//     Box 71 (AT5100-0100)/DRV Statusword/Statusword <-> Data Pointer/Status
//     Box 71 (AT5100-0100)/DRV Target torque/Target torque <-> Data Pointer/Torque
//     Box 71 (AT5100-0100)/DRV Torque actual value/Torque actual value <-> Data Pointer/ActTorque
//     Box 71 (AT5100-0100)/XFB Inputs/Data <-> Data Pointer/HallSensorValues
//   (this object) <-> TcCOM Objects/XTS ProcessingUnit 1/XL Part 2/XL Module 50
//     Box 62 (AT5100-0100)/DRV Commutation angle/Commutation angle <-> Data Pointer/CommutationAngle
//     Box 62 (AT5100-0100)/DRV Controlword/Controlword <-> Data Pointer/Control
//     Box 62 (AT5100-0100)/DRV Statusword/Statusword <-> Data Pointer/Status
//     Box 62 (AT5100-0100)/DRV Target torque/Target torque <-> Data Pointer/Torque
//     Box 62 (AT5100-0100)/DRV Torque actual value/Torque actual value <-> Data Pointer/ActTorque
//     Box 62 (AT5100-0100)/XFB Inputs/Data <-> Data Pointer/HallSensorValues
//   (this object) <-> TcCOM Objects/XTS ProcessingUnit 1/XL Part 2/XL Module 51
//     Box 63 (AT5100-0100)/DRV Commutation angle/Commutation angle <-> Data Pointer/CommutationAngle
//     Box 63 (AT5100-0100)/DRV Controlword/Controlword <-> Data Pointer/Control
//     Box 63 (AT5100-0100)/DRV Statusword/Statusword <-> Data Pointer/Status
//     Box 63 (AT5100-0100)/DRV Target torque/Target torque <-> Data Pointer/Torque
//     Box 63 (AT5100-0100)/DRV Torque actual value/Torque actual value <-> Data Pointer/ActTorque
//     Box 63 (AT5100-0100)/XFB Inputs/Data <-> Data Pointer/HallSensorValues
//   (this object) <-> TcCOM Objects/XTS ProcessingUnit 1/XL Part 2/XL Module 52
//     Box 64 (AT5100-0100)/DRV Commutation angle/Commutation angle <-> Data Pointer/CommutationAngle
//     Box 64 (AT5100-0100)/DRV Controlword/Controlword <-> Data Pointer/Control
//     Box 64 (AT5100-0100)/DRV Statusword/Statusword <-> Data Pointer/Status
//     Box 64 (AT5100-0100)/DRV Target torque/Target torque <-> Data Pointer/Torque
//     Box 64 (AT5100-0100)/DRV Torque actual value/Torque actual value <-> Data Pointer/ActTorque
//     Box 64 (AT5100-0100)/XFB Inputs/Data <-> Data Pointer/HallSensorValues
//   (this object) <-> TcCOM Objects/XTS ProcessingUnit 1/XL Part 2/XL Module 53
//     Box 65 (AT5100-0100)/DRV Commutation angle/Commutation angle <-> Data Pointer/CommutationAngle
//     Box 65 (AT5100-0100)/DRV Controlword/Controlword <-> Data Pointer/Control
//     Box 65 (AT5100-0100)/DRV Statusword/Statusword <-> Data Pointer/Status
//     Box 65 (AT5100-0100)/DRV Target torque/Target torque <-> Data Pointer/Torque
//     Box 65 (AT5100-0100)/DRV Torque actual value/Torque actual value <-> Data Pointer/ActTorque
//     Box 65 (AT5100-0100)/XFB Inputs/Data <-> Data Pointer/HallSensorValues
//   (this object) <-> TcCOM Objects/XTS ProcessingUnit 1/XL Part 2/XL Module 54
//     Box 66 (AT5100-0100)/DRV Commutation angle/Commutation angle <-> Data Pointer/CommutationAngle
//     Box 66 (AT5100-0100)/DRV Controlword/Controlword <-> Data Pointer/Control
//     Box 66 (AT5100-0100)/DRV Statusword/Statusword <-> Data Pointer/Status
//     Box 66 (AT5100-0100)/DRV Target torque/Target torque <-> Data Pointer/Torque
//     Box 66 (AT5100-0100)/DRV Torque actual value/Torque actual value <-> Data Pointer/ActTorque
//     Box 66 (AT5100-0100)/XFB Inputs/Data <-> Data Pointer/HallSensorValues
//   (this object) <-> TcCOM Objects/XTS ProcessingUnit 1/XL Part 2/XL Module 55
//     Box 67 (AT5100-0100)/DRV Commutation angle/Commutation angle <-> Data Pointer/CommutationAngle
//     Box 67 (AT5100-0100)/DRV Controlword/Controlword <-> Data Pointer/Control
//     Box 67 (AT5100-0100)/DRV Statusword/Statusword <-> Data Pointer/Status
//     Box 67 (AT5100-0100)/DRV Target torque/Target torque <-> Data Pointer/Torque
//     Box 67 (AT5100-0100)/DRV Torque actual value/Torque actual value <-> Data Pointer/ActTorque
//     Box 67 (AT5100-0100)/XFB Inputs/Data <-> Data Pointer/HallSensorValues
//   (this object) <-> TcCOM Objects/XTS ProcessingUnit 1/XL Part 2/XL Module 56
//     Box 68 (AT5100-0100)/DRV Commutation angle/Commutation angle <-> Data Pointer/CommutationAngle
//     Box 68 (AT5100-0100)/DRV Controlword/Controlword <-> Data Pointer/Control
//     Box 68 (AT5100-0100)/DRV Statusword/Statusword <-> Data Pointer/Status
//     Box 68 (AT5100-0100)/DRV Target torque/Target torque <-> Data Pointer/Torque
//     Box 68 (AT5100-0100)/DRV Torque actual value/Torque actual value <-> Data Pointer/ActTorque
//     Box 68 (AT5100-0100)/XFB Inputs/Data <-> Data Pointer/HallSensorValues
//   (this object) <-> TcCOM Objects/XTS ProcessingUnit 1/XL Part 2/XL Module 57
//     Box 69 (AT5100-0100)/DRV Commutation angle/Commutation angle <-> Data Pointer/CommutationAngle
//     Box 69 (AT5100-0100)/DRV Controlword/Controlword <-> Data Pointer/Control
//     Box 69 (AT5100-0100)/DRV Statusword/Statusword <-> Data Pointer/Status
//     Box 69 (AT5100-0100)/DRV Target torque/Target torque <-> Data Pointer/Torque
//     Box 69 (AT5100-0100)/DRV Torque actual value/Torque actual value <-> Data Pointer/ActTorque
//     Box 69 (AT5100-0100)/XFB Inputs/Data <-> Data Pointer/HallSensorValues
//   (this object) <-> TcCOM Objects/XTS ProcessingUnit 1/XL Part 3/XL Module 1
//     Box 74 (AT5100-0100)/DRV Commutation angle/Commutation angle <-> Data Pointer/CommutationAngle
//     Box 74 (AT5100-0100)/DRV Controlword/Controlword <-> Data Pointer/Control
//     Box 74 (AT5100-0100)/DRV Statusword/Statusword <-> Data Pointer/Status
//     Box 74 (AT5100-0100)/DRV Target torque/Target torque <-> Data Pointer/Torque
//     Box 74 (AT5100-0100)/DRV Torque actual value/Torque actual value <-> Data Pointer/ActTorque
//     Box 74 (AT5100-0100)/XFB Inputs/Data <-> Data Pointer/HallSensorValues
//   (this object) <-> TcCOM Objects/XTS ProcessingUnit 1/XL Part 3/XL Module 2
//     Box 75 (AT5100-0100)/DRV Commutation angle/Commutation angle <-> Data Pointer/CommutationAngle
//     Box 75 (AT5100-0100)/DRV Controlword/Controlword <-> Data Pointer/Control
//     Box 75 (AT5100-0100)/DRV Statusword/Statusword <-> Data Pointer/Status
//     Box 75 (AT5100-0100)/DRV Target torque/Target torque <-> Data Pointer/Torque
//     Box 75 (AT5100-0100)/DRV Torque actual value/Torque actual value <-> Data Pointer/ActTorque
//     Box 75 (AT5100-0100)/XFB Inputs/Data <-> Data Pointer/HallSensorValues
//   (this object) <-> TcCOM Objects/XTS ProcessingUnit 1/XL Part 3/XL Module 3
//     Box 76 (AT5100-0100)/DRV Commutation angle/Commutation angle <-> Data Pointer/CommutationAngle
//     Box 76 (AT5100-0100)/DRV Controlword/Controlword <-> Data Pointer/Control
//     Box 76 (AT5100-0100)/DRV Statusword/Statusword <-> Data Pointer/Status
//     Box 76 (AT5100-0100)/DRV Target torque/Target torque <-> Data Pointer/Torque
//     Box 76 (AT5100-0100)/DRV Torque actual value/Torque actual value <-> Data Pointer/ActTorque
//     Box 76 (AT5100-0100)/XFB Inputs/Data <-> Data Pointer/HallSensorValues
//   (this object) <-> TcCOM Objects/XTS ProcessingUnit 1/XL Part 3/XL Module 4
//     Box 77 (AT5100-0100)/DRV Commutation angle/Commutation angle <-> Data Pointer/CommutationAngle
//     Box 77 (AT5100-0100)/DRV Controlword/Controlword <-> Data Pointer/Control
//     Box 77 (AT5100-0100)/DRV Statusword/Statusword <-> Data Pointer/Status
//     Box 77 (AT5100-0100)/DRV Target torque/Target torque <-> Data Pointer/Torque
//     Box 77 (AT5100-0100)/DRV Torque actual value/Torque actual value <-> Data Pointer/ActTorque
//     Box 77 (AT5100-0100)/XFB Inputs/Data <-> Data Pointer/HallSensorValues
//   (this object) <-> TcCOM Objects/XTS ProcessingUnit 1/XL Part 3/XL Module 46
//     Box 72 (AT5100-0100)/DRV Commutation angle/Commutation angle <-> Data Pointer/CommutationAngle
//     Box 72 (AT5100-0100)/DRV Controlword/Controlword <-> Data Pointer/Control
//     Box 72 (AT5100-0100)/DRV Statusword/Statusword <-> Data Pointer/Status
//     Box 72 (AT5100-0100)/DRV Target torque/Target torque <-> Data Pointer/Torque
//     Box 72 (AT5100-0100)/DRV Torque actual value/Torque actual value <-> Data Pointer/ActTorque
//     Box 72 (AT5100-0100)/XFB Inputs/Data <-> Data Pointer/HallSensorValues
//   (this object) <-> TcCOM Objects/XTS ProcessingUnit 1/XL Part 3/XL Module 47
//     Box 73 (AT5100-0100)/DRV Commutation angle/Commutation angle <-> Data Pointer/CommutationAngle
//     Box 73 (AT5100-0100)/DRV Controlword/Controlword <-> Data Pointer/Control
//     Box 73 (AT5100-0100)/DRV Statusword/Statusword <-> Data Pointer/Status
//     Box 73 (AT5100-0100)/DRV Target torque/Target torque <-> Data Pointer/Torque
//     Box 73 (AT5100-0100)/DRV Torque actual value/Torque actual value <-> Data Pointer/ActTorque
//     Box 73 (AT5100-0100)/XFB Inputs/Data <-> Data Pointer/HallSensorValues
//   (this object) <-> TcCOM Objects/XTS ProcessingUnit 1/XL Part 3/XL Module 5
//     Box 78 (AT5100-0100)/DRV Commutation angle/Commutation angle <-> Data Pointer/CommutationAngle
//     Box 78 (AT5100-0100)/DRV Controlword/Controlword <-> Data Pointer/Control
//     Box 78 (AT5100-0100)/DRV Statusword/Statusword <-> Data Pointer/Status
//     Box 78 (AT5100-0100)/DRV Target torque/Target torque <-> Data Pointer/Torque
//     Box 78 (AT5100-0100)/DRV Torque actual value/Torque actual value <-> Data Pointer/ActTorque
//     Box 78 (AT5100-0100)/XFB Inputs/Data <-> Data Pointer/HallSensorValues
//   (this object) <-> TcCOM Objects/XTS ProcessingUnit 1/XL Part 3/XL Module 6
//     Box 79 (AT5100-0100)/DRV Commutation angle/Commutation angle <-> Data Pointer/CommutationAngle
//     Box 79 (AT5100-0100)/DRV Controlword/Controlword <-> Data Pointer/Control
//     Box 79 (AT5100-0100)/DRV Statusword/Statusword <-> Data Pointer/Status
//     Box 79 (AT5100-0100)/DRV Target torque/Target torque <-> Data Pointer/Torque
//     Box 79 (AT5100-0100)/DRV Torque actual value/Torque actual value <-> Data Pointer/ActTorque
//     Box 79 (AT5100-0100)/XFB Inputs/Data <-> Data Pointer/HallSensorValues
//   (this object) <-> TcCOM Objects/XTS ProcessingUnit 1/XL Part 3/XL Module 7
//     Box 80 (AT5100-0100)/DRV Commutation angle/Commutation angle <-> Data Pointer/CommutationAngle
//     Box 80 (AT5100-0100)/DRV Controlword/Controlword <-> Data Pointer/Control
//     Box 80 (AT5100-0100)/DRV Statusword/Statusword <-> Data Pointer/Status
//     Box 80 (AT5100-0100)/DRV Target torque/Target torque <-> Data Pointer/Torque
//     Box 80 (AT5100-0100)/DRV Torque actual value/Torque actual value <-> Data Pointer/ActTorque
//     Box 80 (AT5100-0100)/XFB Inputs/Data <-> Data Pointer/HallSensorValues
//   (this object) <-> TcCOM Objects/XTS ProcessingUnit 1/XL Part 3/XL Module 8
//     Box 81 (AT5100-0100)/DRV Commutation angle/Commutation angle <-> Data Pointer/CommutationAngle
//     Box 81 (AT5100-0100)/DRV Controlword/Controlword <-> Data Pointer/Control
//     Box 81 (AT5100-0100)/DRV Statusword/Statusword <-> Data Pointer/Status
//     Box 81 (AT5100-0100)/DRV Target torque/Target torque <-> Data Pointer/Torque
//     Box 81 (AT5100-0100)/DRV Torque actual value/Torque actual value <-> Data Pointer/ActTorque
//     Box 81 (AT5100-0100)/XFB Inputs/Data <-> Data Pointer/HallSensorValues

// ---- DUTs/ST_MoverInfo.TcDUT
TYPE ST_MoverInfo :
STRUCT
	MoverOtcid : otcid;
	PlanarMoverCommandMode : MC_Planar_Mover_Command_Mode;
	State : MC_Planar_State;
	Positition : LREAL;
	Track : Otcid;
	Error: BOOL;
	ErrorID : UDINT;
	TargetTrackPosition  : LREAL;
	TargetTrack : Otcid;
	RemainingDistance : LREAL;
	Gap : LREAL;
	LimitVelo : LREAL; 
	LimitAcc : LREAL;
	LimitDec : LREAL;
	LimitJerk : LREAL;
	
END_STRUCT
END_TYPE

// ---- DUTs/ST_MoverOnTrackInfo.TcDUT
TYPE ST_MoverOnTrackInfo :
STRUCT
	TargetPosition 		: LREAL;
	TargetTrack 		: Otcid;
	Remainingdistance 	: LREAL;
	Gap 				: LREAL;
	LimitV 				: LREAL;
	LimitA 				: LREAL;
	LimitD 				: LREAL;
	LimitJ 				: LREAL;
	GapMode				: MC.MC_GAP_MODE_ON_TRACK;
	DynamicMode			: MC.MC_DYNAMIC_MODE_ON_TRACK;
	Movementtype		: MC.MC_MOVEMENT_TYPE_ON_TRACK;
	
END_STRUCT
END_TYPE

// ---- XlMover/ITFs/I_Mover.TcIO

INTERFACE I_Mover

METHOD CycleUpdate : BOOL
VAR_INPUT
END_VAR
END_METHOD

PROPERTY distToEndOfTrack : Lreal
GET
END_GET
END_PROPERTY

METHOD Init : BOOL
VAR_INPUT
	XtsMover:  I_XtsXlMover1;
	XtsProcessingUnit :  I_XtsProcessingUnit1;
END_VAR
END_METHOD

METHOD JoinNearestTrack : BOOL


VAR

END_VAR
END_METHOD

METHOD LeaveSystemAt : BOOL
VAR_INPUT
	ConnectionOut: REFERENCE TO MC_PlanarTrackConnectionOut;	
END_VAR
END_METHOD

METHOD MoveOnTrack : BOOL
VAR_INPUT
	track: REFERENCE TO MC_PlanarTrack;	
	targetPos: LREAL;
	gap : LREAL; 

END_VAR
END_METHOD

PROPERTY MoverOTCID : OTCID
GET
END_GET
SET
END_SET
END_PROPERTY

PROPERTY MoverStopped : BOOL
GET
END_GET
SET
END_SET
END_PROPERTY

PROPERTY P_Dynamics : REFERENCE TO DynamicConstraint_PathXY;
GET
END_GET
END_PROPERTY

PROPERTY P_IsInitialized : bool
GET
END_GET
END_PROPERTY

PROPERTY P_PlanarFeedback : REFERENCE TO MC_PlanarFeedback
GET
END_GET
END_PROPERTY

PROPERTY P_PlanarMover :   REFERENCE TO  MC_PlanarMover
GET
END_GET
END_PROPERTY

PROPERTY P_SyncFeedback :  REFERENCE TO MC_PlanarFeedbackGearInPosOnTrackWithMasterMover
GET
END_GET
END_PROPERTY

PROPERTY P_TargetTrack : UDINT
GET
END_GET
SET
END_SET
END_PROPERTY

PROPERTY Rework : BOOL
GET
END_GET
SET
END_SET
END_PROPERTY

METHOD SyncToOtherMover : Bool
VAR_INPUT
	masterSyncPos : LREAL; // Position on the master track
	followerSyncPos : LREAL; // position on the follower track
	PlanarMoverToFollow: REFERENCE TO Tc3_Mc3PlanarMotion.MC_PlanarMover;
	masterTrack : REFERENCE TO Tc3_Mc3PlanarMotion.MC_PlanarTrack; 
	followerTrack : REFERENCE TO Tc3_Mc3PlanarMotion.MC_PlanarTrack; 
	velo :  REFERENCE TO LREAL; 
END_VAR
END_METHOD

METHOD  UpdateXtsTrack
VAR_INPUT
END_VAR
VAR

END_VAR
END_METHOD

PROPERTY XlProcessingUnit : I_XtsProcessingUnit1
GET
END_GET
END_PROPERTY

PROPERTY XtsComFeed : REFERENCE TO  XtsCommandFeedback
GET
END_GET
END_PROPERTY

PROPERTY XtsXlMover :  I_XtsXlMover1
GET
END_GET
END_PROPERTY

END_INTERFACE

// ---- POUs/FB_TrackObject.TcPOU
FUNCTION_BLOCK FB_TrackObject
// for a track/part this block keeps a list of the movers in order with their positions on a track

VAR_INPUT
	TrackID: OTCID;
	iMover	:REFERENCE TO ARRAY[1..nMoverCount] OF I_Mover;
END_VAR

VAR_OUTPUT
	bBusy: BOOL;
	bDone: BOOL;
	bError: BOOL;
	bInit: BOOL;
	ipResultMessage: I_TcMessage := fbResult;
	moverIDs : ARRAY[1..nMoverCount] OF UDINT;
	
END_VAR

VAR_STAT
	nNumMoversOnTrack: UDINT; //numberofMovers currently on this track
	nMoverList: ARRAY [1..nMoverCount] OF OTCID; //list of movers currently on the track 
	
	Moverdist: ARRAY[1..nMoverCount] OF LREAL;
	MoverPos: ARRAY[1..nMoverCount] OF LREAL;
	
	
END_VAR

VAR

	fbResult: FB_TcMessage;
	_ipComObject: ITComObject;
	PID_MOverList				: PTCID := 16#05030149;
	PID_NumMover				: PTCID := 16#050300C5;
END_VAR

IF NOT bInit THEN
	IF GetComObject(nObjectId:=TrackID) THEN
		bInit:=TRUE;
	END_IF
	RETURN;
END_IF

METHOD CyclicUpdate : BOOL
VAR_INPUT
END_VAR

VAR_INST
	J: UDINT;
	I: UINT;
END_VAR
IF bInit THEN 
	GetNumMovers(); 
	GetMoverList(); 
END_IF 
MEMSET(ADR(moverIDs),0,SIZEOF(moverIDs)); // have to clear the list 
MEMSET(ADR(Moverdist),0,SIZEOF(Moverdist)); // have to clear the list 
MEMSET(ADR(MoverPos),0,SIZEOF(MoverPos)); // have to clear the list 
FOR J := 1 TO nNumMoversOnTrack DO  
	FOR I := 1 TO nNumMovers DO  
		IF iMover[I].MoverOTCID = nMoverList[J] THEN 
			moverIDs[J] := I; 
		END_IF
	END_FOR

	
END_FOR

FOR J := 1 TO nNumMoversOnTrack DO  
	
	IF J < nNumMoversOnTrack - 1 THEN 
		 IF fbMover[moverIDs[j+1]].distToEndOfTrack - fbMover[moverIDs[j]].distToEndOfTrack > 0 THEN 
			Moverdist[j]:= fbMover[moverIDs[j+1]].distToEndOfTrack - fbMover[moverIDs[j]].distToEndOfTrack;
		ELSE
			Moverdist[j]:=-1;	
		END_IF
		MoverPos[j]:= fbMover[moverIDs[j+1]].distToEndOfTrack; // folowwing movers distance 
		//idist := fbMover[moverIDs[I]].distToEndOfTrack; //this movers distance 
	END_IF
	
END_FOR
END_METHOD

METHOD findMergePosition : BOOL
VAR_INPUT
	mergeSyncCommandPos : LREAL;
	spaceToMerge :LREAL; 
END_VAR
VAR_OUTPUT 
	nMoverToFollow: UDINT; 
	mergeWithoutFollow : BOOL; 
	mergeNotPossible : BOOL; 
END_VAR
VAR_INST 
	I: UDINT;
	moverInMerge: UDINT;
	moverIsWhereWeSync: BOOL;
	moversDist: LREAL;
	Iplus1Dist: LREAL;
	idist: LREAL;

	needToFollow: BOOL;

END_VAR
mergeNotPossible := TRUE; 
mergeWithoutFollow:=FALSE;
nMoverToFollow := 0; 
moverInMerge := 0;
needToFollow := TRUE;  
IF nNumMoversOnTrack = 0  THEN // if there's no movers on the track we can just merge 
	mergeWithoutFollow := TRUE;
	mergeNotPossible := FALSE; 
ELSE
  	// there's movers in the track we need to look where there are 
	// go through the movers positions and find a place to merge if available 
	FOR I := 1 TO nNumMoversOnTrack DO 
		// is this mover in the range where we would sync? 
		moverIsWhereWeSync := IsBetween(fbMover[moverIDs[I]].distToEndOfTrack, mergeSyncCommandPos, mergeSyncCommandPos + spaceToMerge); 
		needToFollow := IsBetween(fbMover[moverIDs[I]].distToEndOfTrack, mergeSyncCommandPos, mergeSyncCommandPos + spaceToMerge); //lagerwindow we can merge but must sync still
		IF moverIsWhereWeSync THEN //if the mover is where we would sync start looking for places to merge behind it
			moverInMerge := moverIDs[I]; // this mover is is the id of the mover thats in the way 
			// can we merge behind this one ?
			IF I < nNumMoversOnTrack THEN 
		//		Moverdist[i+10]:=moversDist := fbMover[moverIDs[I+1]].distToEndOfTrack - fbMover[moverIDs[I]].distToEndOfTrack;
	//			Moverdist[i]:=Iplus1Dist := fbMover[moverIDs[I+1]].distToEndOfTrack; // folowwing movers distance 
	//			idist := fbMover[moverIDs[I]].distToEndOfTrack; //this movers distance 
				// is the spacing between these two movers bigger than the space we need to merge?
				IF (Moverdist[i] )> spaceToMerge THEN 
					nMoverToFollow := moverIDs[I]; //yes follow this mover 
					mergeNotPossible := FALSE; // the merge is possible 
					EXIT; 
				END_IF
			ELSIF I = nNumMoversOnTrack THEN // this is the last mover 
				// look how much space is behind this mover that is bigger than the merge gap, merge behind this mover
				IF fbMover[moverIDs[I]].distToEndOfTrack < mergeSyncCommandPos+spaceToMerge THEN // the mover is far enough along to sync to it.
					nMoverToFollow := moverIDs[I]; //yes follow this mover 
					mergeNotPossible := FALSE; // the merge is possible 
				END_IF  
			END_IF	
		END_IF
	END_FOR 
	//if we went through the whole list and no mover is in the range where we would merge in, then just merge 
	IF fbMover[moverIDs[1]].distToEndOfTrack > 6000 THEN //there's noone where we want to merge, just merge in 
		mergeWithoutFollow:=TRUE;
		mergeNotPossible := FALSE;
	END_IF
END_IF
IF mergeNotPossible THEN 
	nMoverToFollow := 0; 
END_IF
END_METHOD

METHOD GetComObject : BOOL
VAR_INPUT
	nObjectId: OTCID;
END_VAR
IF FW_ObjMgr_GetObjectInstance(	oid		:= nObjectId, 
								iid		:= TC_GLOBAL_IID_LIST.IID_ITComObject, 
								pipUnk	:= ADR(_ipComObject)) = 0
THEN
	GetComObject := TRUE;
END_IF
END_METHOD

METHOD GetMoverList : BOOL
VAR
	nData 			: UDINT := SIZEOF(nMoverList);
	pData 			: PVOID := ADR(nMoverList);
	stEventEntry	: TcEventEntry;
	pstEventEntry	: REFERENCE TO TcEventEntry REF= stEventEntry;
END_VAR
VAR_INST
	hResult : HRESULT;
END_VAR
bError := FALSE;

IF _ipComObject <> 0 THEN 
	 hResult := 	_ipComObject.TcgetObjPara(		pid := PID_MOverList,
													nData := nData,
													pData := pData,
													pgp := 0); 	
	IF hResult = 0 THEN
		GetMoverList := TRUE;
	ELSE
		HRESULTAdsErr_TO_TcEventEntry(hResult,stEventEntry);
		IF NOT fbResult.EqualsToEventEntryEx( stOther := stEventEntry) THEN
			fbResult.CreateEx(stEventEntry, 0);
			fbResult.Send(0);
			fbResult.Release();
		END_IF
		bError := TRUE;
	END_IF							
END_IF
END_METHOD

METHOD GetNumMovers : BOOL
VAR
	stEventEntry: TcEventEntry;
	pstEventEntry: REFERENCE TO TcEventEntry := stEventEntry;
	nData 			: UDINT := SIZEOF(nNumMoversOnTrack);
	pData 			: PVOID := ADR(nNumMoversOnTrack);
END_VAR

VAR_INST
	hResult : HRESULT;
END_VAR
bError := FALSE;

IF _ipComObject <> 0 THEN 	
	

	 hResult := 	_ipComObject.TcGetObjPara(		pid := PID_NumMover,
													nData := nData,
													pData := pData,
													pgp := 0); 	
	IF hResult = 0 THEN
		GetNumMovers := TRUE;
	ELSE
		HRESULTAdsErr_TO_TcEventEntry(hResult,stEventEntry);
		IF NOT fbResult.EqualsToEventEntryEx( stOther := stEventEntry) THEN
			fbResult.CreateEx(stEventEntry, 0);
			fbResult.Send(0);
			fbResult.Release();
		END_IF
		bError := TRUE;
	END_IF							
END_IF
END_METHOD

END_FUNCTION_BLOCK

// ---- POUs/MAIN.TcPOU
PROGRAM MAIN
VAR
	RuntimeDuration	: STRING;
	TempRuntimeDur	: TIME;
	RuntimeTimer	: TON;
	CurrentSysTime	: ULINT;

	bAllDone		: BOOL;
	bStopSequence	: BOOL;
	HMI_StopCmd		: BOOL;
	
	nCase 		: INT;
	nMoveState		: ARRAY[1..nMoverCount] OF INT;
	

	
	nForCounter: UDINT;
	M,N,T,Tr : UINT;
//	slowDynamics: DynamicConstraint_PathXY;
	haltDynamics : DynamicConstraint_PathXY;
	stopAndWait : ARRAY[1..GVL_Mc.nMoverCount] OF TON; 
	waitForGapParkPos: LREAL := 3500;
	// Magnet
	MagnetValue AT%Q*: INT;
	MagnetFdbkValue AT%I* : INT;
	bMagnetOn : BOOL;
	MagnetOnManHMICmd 	: BOOL;
	tMagnetOnTime	: TIME := T#3S;

	Init : BOOL ; 	
	
	IsMoverCommandedInShortcut: BOOL;
	IsMoverInBlockingArea: BOOL;
	nActStopPos: UINT := 1;
	Fp_error : R_Trig;

	Switch : BOOL;
	WithoutSwitch : BOOL := TRUE;
	SwtichOnly: BOOL;
	
	MoverStop 	AT%I* :BOOL;
	MoverStopDone AT%Q*		: BOOL;
	Info 		AT%Q*: BOOL;
	Operating	AT%Q*: BOOL;
	Process		AT%Q*: BOOL;
	Fault		AT%Q*: BOOL;
	Emergency	AT%Q*: BOOL;
	
	Voltage1 AT%I*: UDINT;
	Voltage2 AT%I*: UDINT;
	
	
	TcRestart : TC_Restart;
	Restart : BOOL;
	busy : BOOL;
	rt_InitStart : R_TRIG;
	rt_InitStop : R_TRIG;
	bStartSequence: BOOL;
	
	FP_Counter : r_trig;
	Switchcounter : DINT;
	test : LREAL;
	Horntimer : tp; 
	R_trigHorn : R_trig;
	
	TestPowerMat : BOOL := TRUE;
	StopTime : TIME := T#1S;
	StopTimer :ARRAY[1..nMoverCount] OF ton;
	StartTimer :ARRAY[1..nMoverCount] OF BOOL;
	
	
	MoverPos :ARRAY[1..nMoverCount] OF PositionXYC;
	ArcLength :ARRAY[1..nMoverCount] OF LREAL;
	TrackPos :ARRAY[1..nMoverCount] OF ARRAY[1..nMoverCount] OF PositionXYC;
	
	//searchGap : F_SearchTheBigTrackForAHole; 
	aMoverTrack : ARRAY[1..nMoverCount] OF Global.OTCID;
	FirstMoverTrackPos : LREAL;
	MoverGap : LREAL;
	FTrigTrackCount : F_Trig;
	MoverNo  : UDINT;
	stMoverConfigSlow	: ST_MoverConfig;
	stMoverConfigNormal : ST_MoverConfig;
	stMoverConfigFast  : ST_MoverConfig;
	stMoverCfgAggressive : ST_MoverConfig;
	stMoverCfgHalt : ST_MoverConfig;
	
	stMergeConfig		 : ST_MergeConfig;
	SwitchConfig		 : ST_SwitchConfig;
	
	SwitchStatus 		  : ST_SwitchStatus;

	ModuleState1 AT%I*: E_EcState;
	ModuleState2 AT%I*: E_EcState;
	ModuleState3 AT%I*: ARRAY[0..2] OF E_EcState;
	
	MessageTrigger : ARRAY[1..20] OF R_trig;
	
	//========= Merge =========================================
	
	SwitchParkPos : LREAL := 3500;
	nextMoverForSwitch: UDINT :=1;
	moverInSwitchDoNotSendAnother: BOOL;
	trapError: BOOL;
	trapErrorID: UDINT;
	moverWithFault: UDINT;
	stepWithFault: INT;
	
	followSyncPos: LREAL;
	masterSyncPos: LREAL;
	masterPosAtSync: LREAL;
	followerPosAtSync: LREAL;
	moverInFront: UDINT;
	gapStart: LREAL := 8500; //5600
	gapLength: LREAL := 2200; //1800
	fbTrackobject : FB_TrackObject;
	getList: BOOL;
	directMerge: BOOL;
	mergeNotPossible: BOOL;
	
	endOfBigTrack : LREAL; 
	endOfSmallTrack : LREAL; 
	endOfMainTrack : LREAL; 
	followerToEndOfTrack: LREAL;
	leaderToEndofTrack: LREAL;
	distToMoverInFront: LREAL;
	moverSwitching: UDINT;
	switchingMoverPosition: LREAL;
	trapWhenMagnetturnedOn: R_TRIG;
	moverPositionWhenMagnetTurnedOn: LREAL;
	moverInSwitch: UDINT;
END_VAR


// =====================
// Initalize XTS Utility
GVL_MC.fbXtsEnvironment.Init(GVL_MC.cmdFeedback);
IF NOT GVL_MC.cmdFeedback.IsDone THEN
	RETURN;
END_IF
//*****************************************************
Emergency :=  MoverStop;

Operating := NOT  MoverStop;

//================== Check Voltage=====================================================
R_trigHorn(clk := Voltage1< 250000 );
//Horntimer(in:= ( R_trigHorn.Q ) , PT:= T#2S,Q=> info);
IF R_trigHorn.Q THEN
	ADSLOGSTR(msgCtrlMask:= ADSLOG_MSGTYPE_LOG , msgFmtStr:= 'Module Voltage Fault ' , strArg:= '');
END_IF 
//=================== Check State of Modules===========================================

MessageTrigger[1](clk:=ModuleState1 <> 8 AND nCASE> 0);
IF MessageTrigger[1].Q THEN
	ADSLOGSTR(msgCtrlMask:= ADSLOG_MSGTYPE_LOG , msgFmtStr:= 'Module Fault Line 1 %s' , strArg:= TO_STRING(ModuleState1));
END_IF

MessageTrigger[2](clk:=ModuleState2 <> 8 AND nCASE> 0);
IF MessageTrigger[2].Q THEN
	ADSLOGSTR(msgCtrlMask:= ADSLOG_MSGTYPE_LOG , msgFmtStr:= 'Module Fault Line 2 %s ' , strArg:= TO_STRING(ModuleState2));
END_IF

MessageTrigger[3](clk:=ModuleState3[0] <> 8 AND nCASE> 0);
IF MessageTrigger[3].Q THEN
	ADSLOGSTR(msgCtrlMask:= ADSLOG_MSGTYPE_LOG , msgFmtStr:= 'Module Fault Line 3 Default SyncUnit %s ' , strArg:= TO_STRING(ModuleState3[0]));
END_IF

MessageTrigger[4](clk:=ModuleState3[1] <> 8 AND nCASE> 0);
IF MessageTrigger[4].Q THEN
	ADSLOGSTR(msgCtrlMask:= ADSLOG_MSGTYPE_LOG , msgFmtStr:= 'Module Fault Line 3 XtsTask SyncUnit %s ' , strArg:= TO_STRING(ModuleState3[1]));
END_IF

MessageTrigger[5](clk:=ModuleState3[2] <> 8 AND nCASE> 0);
IF MessageTrigger[5].Q THEN
	ADSLOGSTR(msgCtrlMask:= ADSLOG_MSGTYPE_LOG , msgFmtStr:= 'Module Fault Line 3 PlcTask SyncUnit %s ' , strArg:= TO_STRING(ModuleState3[2]));
END_IF

//=====================================================================================

IF nCASE > 90 THEN
	Process := TRUE;
ELSE 
	Process := FALSE;	
END_IF

IF NOT MoverStop AND NOT MoverStopDone AND (nCase = 100) THEN
	ADSLOGSTR(msgCtrlMask:= ADSLOG_MSGTYPE_LOG , msgFmtStr:= 'E-Stop ' , strArg:= '');
	FOR nForCounter:=1 TO nNumMovers DO
		fbMover[nForCounter].P_Dynamics.SetValuesVADJ(stMoverConfigNormal.velo,stMoverConfigNormal.Accel,stMoverConfigNormal.Decel,stMoverConfigNormal.Jerk);
		nCase := 140;
	END_FOR		
ELSIF 	MoverStop THEN
	MoverStopDone := FALSE;
END_IF



TcRestart(
NETID:= '', 
RESTART:= Restart OR (GVL_Mc.HWStart AND NOT GVL_Mc.HWStop), 
TMOUT:=T#5S , 
BUSY=>busy , 
ERR=> , 
ERRID=> );

CurrentSysTime	:= Tc2_System.F_GetSystemTime();

IF TcRestart.BUSY THEN
	RuntimeTimer.IN 	:= FALSE;
ELSIF Process THEN
	RuntimeTimer.IN		:= TRUE;
	TempRuntimeDur		:= RuntimeTimer.ET;
	RuntimeDuration		:= TIME_TO_STRING(TempRuntimeDur);
END_IF
RuntimeTimer(PT := T#7D);

rt_InitStart(clk:= (bStartSequence OR GVL_Mc.HWStart) AND GVL_Mc.HWStop);
IF rt_InitStart.Q THEN
	nCase := 10;
	bStartSequence	:= FALSE;

	stMoverConfigSlow.Velo := 1000;
// 	stMoverConfigSlow.Accel := 4000;
// 	stMoverConfigSlow.Decel := 4000; 
// 	stMoverConfigSlow.Jerk := 16000;
	stMoverConfigFast.Velo := 4000;
// 	stMoverConfigFast.Accel := 4000;
// 	stMoverConfigFast.Decel := 4000; 
// 	stMoverConfigFast.Jerk := 16000;
	stMoverCfgHalt.Decel := 2000; 
	stMoverCfgHalt.Jerk := 10000;
	
//	slowDynamics.SetValuesVADJ(stMoverConfigSlow.Velo,stMoverConfigSlow.Accel,stMoverConfigSlow.Decel,stMoverConfigSlow.Jerk);
//	fastDynamics.SetValuesVADJ(stMoverConfigFast.Velo,stMoverConfigFast.Accel,stMoverConfigFast.Decel,stMoverConfigFast.Jerk);
	haltDynamics.SetValuesVADJ(stMoverCfgHalt.Velo,stMoverCfgHalt.Accel,stMoverCfgHalt.Decel,stMoverCfgHalt.Jerk);
END_IF
haltDynamics.SetValuesVADJ(stMoverCfgHalt.Velo,stMoverCfgHalt.Accel,stMoverCfgHalt.Decel,stMoverCfgHalt.Jerk);
GVL_Mc.StartLight := MoverStop AND nCase < 100;
GVL_Mc.StopLight  := (nCase = 100);

IsMoverInBlockingArea := FALSE;

FOR M := 1 TO GVL_Mc.nNumMovers DO///Movers
	StopTimer[M](in:=StartTimer[m],PT:=StopTime);

	
	IF NOT GVL_MC.fbMover[GVL_Mc.nNumMovers].P_IsInitialized THEN
		GVL_MC.ipXtsProcessingUnit :=  GVL_MC.fbXtsEnvironment.ProcessingUnit(1,0);
		GVL_MC.ipXlMover  :=  GVL_MC.fbXtsEnvironment.ProcessingUnit(1, 0).XlMover(m, 0);
		GVL_MC.fbMover[m].Init( GVL_MC.ipXlMover, GVL_MC.ipXtsProcessingUnit); 
		iMover[m] := fbMover[m] ;
	END_IF
	 MoverFeedback[m].Update();
	GVL_MC.fbMover[m].CycleUpdate();
	
	GVL_Mc.Mover[M].MoverPos  :=GVL_MC.fbMover[M].P_PlanarMover.MCTOPLC.SETONTRACK.SetPos;
	GVL_Mc.Mover[M].TrackID:= GVL_MC.fbMover[M].P_PlanarMover.MCTOPLC.SETONTRACK.TrackOID;
	GVL_Mc.Mover[M].MoverNumber := M;
		
	TR := Tr+1;
	IF Tr = 4 THEN
		Tr :=1;
	END_IF
	ArcLength[M] :=GVL_Mc.MC_Tracks[Tr].GetArcLengthClosestTo(MoverPos[M]);
	GVL_Mc.MC_Tracks[Tr].GetPositionAt(ArcLength[M],TrackPos[M][Tr]);
	
	IF ABS(MoverPos[m].x - TrackPos[M][Tr].x) < 1 AND  ABS(MoverPos[m].y - TrackPos[M][Tr].y) < 1 THEN
 		GVL_Mc.Mover[M].MoverTrackNr := Tr;
	END_IF	
	
	IsMoverInBlockingArea := IsMoverInBlockingArea OR (Mover[M].TrackID = GVL_Mc.MC_Tracks[E_TrackNum.main].MCTOPLC_STD.TrackOID AND IsBetween(Mover[M].MoverPos, SwitchConfig.MagnetStartPosition - 100, SwitchConfig.MagnetEndPosition + 100));

	Fp_error(clk := GVL_MC.fbMover[M].P_PlanarMover.Error AND GVL_MC.fbMover[M].XtsXlMover.GetIsActive(0) AND nCASE = 100);
	IF Fp_error.Q THEN
		nCase := 140;
		Fault := TRUE;
		bMagnetOn := FALSE;
		ADSLOGSTR(msgCtrlMask:= ADSLOG_MSGTYPE_LOG , msgFmtStr:= 'Mover %s Faulted ' , strArg:= INT_TO_STRING(M));
	ELSE
		Fault := FALSE;
	END_IF
	
	IF aMoverTrack[1] <> 0 AND_THEN GVL_MC.fbMover[M].P_PlanarMover.MCTOPLC.STD.MoverOID = aMoverTrack[1] THEN
		FirstMoverTrackPos := GVL_MC.fbMover[M].P_PlanarMover.MCTOPLC.SETONTRACK.SetPos;
	END_IF
	
END_FOR

FOR T := 1 TO nTrackCount DO 
	MC_Tracks[T].Update();
	MC_Trackfeedback[T].Update();
	
END_FOR
 MoverGap := (GVL_Mc.MC_Tracks[E_TrackNum.Big].GetLength()- FirstMoverTrackPos);
 
//================  merge ===============

fbTrackobject(TrackID:= MC_Tracks[E_TrackNum.big].MCTOPLC_STD.TrackOID,iMover:= iMover,trackLength:= GVL_Mc.MC_Tracks[E_TrackNum.Big].GetLength()); 
fbTrackobject.CyclicUpdate(); 


//======================================

CASE nCase OF
	10:
		
		Fault := FALSE;
		nCase := 20;

	20:
		FOR T := 1 TO nTrackCount DO 
			MC_Tracks[T].Enable(MC_Trackfeedback[T]);
		END_FOR
				nCase := 30;
				
	30: 
		IF MC_Trackfeedback[1].Done AND MC_Trackfeedback[2].Done AND MC_Trackfeedback[3].Done THEN
			nCase := 35;
		END_IF
		
		
	35:
		FOR nForCounter:=1 TO nNumMovers DO
			GVL_MC.fbMover[nForCounter].P_Dynamics.SetValuesVADJ(stMoverConfigNormal.velo,stMoverConfigNormal.Accel,stMoverConfigNormal.Decel,stMoverConfigNormal.Jerk);
			fbMover[nForCounter].P_PlanarMover.Reset(MoverFeedback[nForCounter]);
		END_FOR
		nCase := 36;	
			
	36:	
		bAllDone:=TRUE;
		FOR nForCounter:=1 TO nNumMovers DO
			bAllDone:=bAllDone AND MoverFeedback[nForCounter].Done;
		END_FOR
		
		IF bAllDone THEN
			nCase := 40;
		END_IF
				
	40:
		FOR nForCounter:=1 TO nNumMovers DO
			fbMover[nForCounter].P_PlanarMover.Enable(MoverFeedback[nForCounter]);
		END_FOR
		nCase := 50;
			
	50:
		bAllDone:=TRUE;
		FOR nForCounter:=1 TO nNumMovers DO
			bAllDone:=bAllDone AND MoverFeedback[nForCounter].Done;
		END_FOR
		
		IF bAllDone THEN
			nCase := 60;
		END_IF

	60:
		FOR nForCounter:=nNumMovers TO 1  BY -1 DO
			fbMover[nForCounter].JoinNearestTrack();
		END_FOR
		
		nCase := 70;
		
		
	70:
		bAllDone:=TRUE;
		FOR nForCounter:=1 TO nNumMovers DO
			bAllDone:=bAllDone AND fbMover[nForCounter].P_PlanarFeedback.Done;
		END_FOR
		
		IF bAllDone THEN
			nCase := 80;
		END_IF
		
	80:	
		FOR nForCounter:=1 TO nNumMovers DO
			nMoveState[nForCounter] := 0;
		END_FOR
		
		nCase := 100;

	100:
		
		FOR nForCounter:=1 TO nNumMovers DO
			fbMover[nForCounter].P_Dynamics.SetValuesVADJ(stMoverConfigNormal.velo,stMoverConfigNormal.Accel,stMoverConfigNormal.Decel,stMoverConfigNormal.Jerk);
			IF MoverNo <> 0 AND_THEN 	fbMover[MoverNo].P_PlanarMover.MCTOPLC.SETONTRACK.TrackOID =	 GVL_Mc.MC_Tracks[E_TrackNum.Big].MCTOPLC_STD.TrackOID THEN
				IsMoverCommandedInShortcut := FALSE;
			//	MoverNo := 0;
			END_IF
			
			//Adjust the first mover parameters to induce a platoon
			fbMover[1].P_Dynamics.SetValuesVADJ(V:= stMoverConfigNormal.velo-stMoverConfigNormal.VeloComp, A:= stMoverConfigNormal.Accel, D:= stMoverConfigNormal.Decel, J:= stMoverConfigNormal.Jerk);	
			
			IF SwitchConfig.DivertConfig.MaxAllowedDivertCount > 0 THEN
				WithoutSwitch 	:= FALSE;
			ELSE
				WithoutSwitch	:= TRUE;
			END_IF
			
			CASE nMoveState[nForCounter] OF
				
				0: // Track 3 Main Cycle
					fbMover[nForCounter].P_Dynamics.SetValuesVADJ(stMoverConfigNormal.velo,stMoverConfigNormal.Accel,stMoverConfigNormal.Decel,stMoverConfigNormal.Jerk);
					fbMover[nForCounter].MoveOnTrack(track:= GVL_Mc.MC_Tracks[E_TrackNum.Main], targetPos:= GVL_Mc.MC_Tracks[E_TrackNum.Main].GetLength()-500, gap:= stMoverConfigNormal.MoverGap);
				
					nMoveState[nForCounter] := 10;
					
				10:
					IF Mover[nForCounter].MoverPos > GVL_Mc.MC_Tracks[E_TrackNum.Main].GetLength()-6000  AND  Mover[nForCounter].TrackID =   GVL_Mc.MC_Tracks[E_TrackNum.Main].MCTOPLC_STD.TrackOID    THEN//     MCTrackOid_MainSemicircle THEN
						IF  (SwtichOnly OR NOT IsMoverCommandedInShortcut )AND NOT WithoutSwitch  AND  nForCounter = nextMoverForSwitch THEN // AND NOT( moverInSwitchDoNotSendAnother)  THEN
							nMoveState[nForCounter] := 40; // 20 - BigCycel
								moverInSwitchDoNotSendAnother := TRUE; 
							//IF fbPlanarMover[nForCounter].IsCommandedInShortcut THEN
								IsMoverCommandedInShortcut := TRUE;
								MoverNo :=nForCounter; /// fbPlanarMover[nForCounter].McPlanarMover.MCTOPLC.STD.MoverOID;
								IF nextMoverForSwitch >= nNumMovers THEN // send the next mover to the switch
									nextMoverForSwitch := 1; 
								ELSE 
									nextMoverForSwitch := nextMoverForSwitch + 1; 
								END_IF
							//END_IF
						ELSE
							nMoveState[nForCounter] := 20;  // 40- SmallCycel					
						END_IF
					END_IF

				
				20:
					fbMover[nForCounter].P_Dynamics.SetValuesVADJ(stMoverConfigNormal.velo,stMoverConfigNormal.Accel,stMoverConfigNormal.Decel,stMoverConfigNormal.Jerk);
					fbMover[nForCounter].MoveOnTrack(track:= GVL_Mc.MC_Tracks[E_TrackNum.Big], targetPos:= GVL_Mc.MC_Tracks[E_TrackNum.Big].GetLength()-1000, gap:= stMoverConfigNormal.MoverGap);
			
					nMoveState[nForCounter] := 30;
				
					
				30:
					IF fbMover[nForCounter].P_PlanarFeedback.Error AND NOT trapError THEN //trap the error once.  
						moverWithFault := nForCounter; 
						trapError := fbMover[nForCounter].P_PlanarFeedback.Error; 
						trapErrorID := fbMover[nForCounter].P_PlanarFeedback.ErrorId; 
						stepWithFault := 30; 
					END_IF 
					IF Mover[nForCounter].MoverPos > GVL_Mc.MC_Tracks[E_TrackNum.Big].GetLength()-12000 AND  Mover[nForCounter].TrackID = GVL_Mc.MC_Tracks[E_TrackNum.big].MCTOPLC_STD.TrackOID    THEN//      MCTrackOid_BigSemicircle THEN
						nMoveState[nForCounter] := 0;
					END_IF				
				
			
				40:
					fbMover[nForCounter].P_Dynamics.SetValuesVADJ(stMoverConfigNormal.velo,stMoverConfigNormal.Accel,stMoverConfigNormal.Decel,stMoverConfigNormal.Jerk);
					fbMover[nForCounter].MoveOnTrack(track:= GVL_Mc.MC_Tracks[E_TrackNum.Small], targetPos:= SwitchParkPos, gap:= stMoverConfigNormal.MoverGap);
					
					nMoveState[nForCounter] := 45;
	
				45: 
					IF fbMover[nForCounter].P_PlanarFeedback.Error AND NOT trapError THEN //trap the error once.   
						trapError := fbMover[nForCounter].P_PlanarFeedback.Error; 
						trapErrorID := fbMover[nForCounter].P_PlanarFeedback.ErrorId;
						stepWithFault := 45;
 						moverWithFault := nForCounter; 
					END_IF
					IF fbMover[nForCounter].P_PlanarFeedback.Done THEN 
						nMoveState[nForCounter] := 50; //50;
						stopAndWait[nForCounter](IN:=TRUE, PT:=StopTime); 
					END_IF 	

				50:
					stopAndWait[nForCounter](); 
					IF stopAndWait[nForCounter].Q  OR NOT TestPowerMat THEN // send the mover to a sync Position 2.6m before the end of the track 
						stopAndWait[nForCounter](IN:=FALSE); 							
					//	fbMover[nForCounter].P_Dynamics.SetValuesVADJ(stMoverConfigNormal.velo,stMoverConfigNormal.Accel,stMoverConfigNormal.Decel,stMoverConfigNormal.Jerk);
					//	fbMover[nForCounter].MoveOnTrack( GVL_Mc.MC_Tracks[E_TrackNum.Small], GVL_Mc.MC_Tracks[E_TrackNum.Small].GetLength()-waitForGapParkPos,stMoverConfigNormal.MoverGap,stMoverConfigNormal.velo);
					//	searchGap(resetSearch:=TRUE, fbMover := fbMover); 
						nMoveState[nForCounter] := 60; 
					END_IF 
					
				60: // look for a merge position 
					//IF fbMover[nForCounter].P_PlanarFeedback.Done THEN// MCTrackOid_Shortcut THEN
							fbTrackobject.findMergePosition(
								mergeSyncCommandPos := gapStart , 
								spaceToMerge := gapLength, 
								nMoverToFollow => moverInFront, 
								mergeWithoutFollow => directMerge, 
								mergeNotPossible => mergeNotPossible); 
							IF directMerge OR  ( moverInFront <> 0) AND NOT mergeNotPossible THEN
								nMoveState[nForCounter] := 70;
							END_IF 
				//	END_IF
				70:  //merge with gap zero
					//issue commmand to sync 
					IF  directMerge THEN 
						fbMover[nForCounter].P_Dynamics.SetValuesVADJ(stMoverConfigNormal.velo,stMoverConfigNormal.Accel,stMoverConfigNormal.Decel,stMoverConfigNormal.Jerk);
						fbMover[nForCounter].MoveOnTrack(track:= GVL_Mc.MC_Tracks[E_TrackNum.Main], targetPos:= GVL_Mc.MC_Tracks[E_TrackNum.Main].GetLength()-500, gap:= stMoverConfigNormal.MoverGap);

						nMoveState[nForCounter] := 10; 
					ELSIF moverInFront <>0 THEN 
						fbMover[nForCounter].P_Dynamics.SetValuesVADJ(stMoverConfigNormal.velo,stMoverConfigNormal.Accel,stMoverConfigNormal.Decel,stMoverConfigNormal.Jerk);
						masterSyncPos := GVL_Mc.MC_Tracks[E_TrackNum.Big].GetLength()-2500;
						masterPosAtSync := Mover[moverInFront].MoverPos; 
						followSyncPos := GVL_Mc.MC_Tracks[E_TrackNum.Small].GetLength()-stMoverConfigNormal.MoverGap-2500;
						followerPosAtSync :=Mover[nForCounter].MoverPos; 
						fbMover[nForCounter].SyncToOtherMover( 
							masterSyncPos := masterSyncPos,
							masterTrack := GVL_Mc.MC_Tracks[E_TrackNum.Big],
							followerSyncPos := followSyncPos,
							followerTrack := GVL_Mc.MC_Tracks[e_TrackNum.Small],
							PlanarMoverToFollow := fbMover[moverInFront].P_PlanarMover,
							velo:= stMoverConfigNormal.velo);
							nMoveState[nForCounter] := 80; 
						// reduce the gap of the leading mover 
						fbMover[moverInFront].MoveOnTrack(track:= GVL_Mc.MC_Tracks[E_TrackNum.Main], targetPos:= GVL_Mc.MC_Tracks[E_TrackNum.Main].GetLength()-500, gap:= 0);

					END_IF 
					
				80: // wait for in Sync 
					IF fbMover[nForCounter].P_SyncFeedback.Active AND MOver[moverInFront].TrackID =  GVL_Mc.MC_Tracks[E_TrackNum.Big].MCTOPLC_STD.TrackOID THEN // actively syncing calculate distance from mover 
						followerToEndOfTrack := fbMover[nForCounter].distToEndOfTrack; 
						leaderToEndofTrack := fbMover[moverInFront].distToEndOfTrack; 
						distToMoverInFront := followerToEndOfTrack - leaderToEndofTrack; 
					ELSE 
						followerToEndOfTrack := 0; 
						leaderToEndofTrack := 0; 
						distToMoverInFront := 0;
					END_IF
					IF fbMover[nForCounter].P_SyncFeedback.inSync OR  MOver[nForCounter].TrackID =  GVL_Mc.MC_Tracks[E_TrackNum.Main].MCTOPLC_STD.TrackOID THEN 
						nMoveState[nForCounter] := 10;
						IsMoverCommandedInShortcut :=FALSE;
					ELSIF	fbMover[nForCounter].P_SyncFeedback.Error THEN
						nMoveState[nForCounter] := 60;
					END_IF 
					
				END_CASE
		
		END_FOR

		rt_InitStop(CLK := HMI_StopCmd OR NOT GVL_Mc.HWStop);
		IF rt_InitStop.Q AND NOT bStopSequence THEN
			bStopSequence := TRUE;
		END_IF
		IF bStopSequence AND NOT(IsMoverInBlockingArea) THEN
			nCase := 110;
			bStopSequence := FALSE;
		END_IF
		
		110:
			N:= nNumMovers;
			FOR nForCounter:=1 TO nNumMovers DO		
				aStopPositions[nForCounter] := fbMover[nForCounter].XtsXlMover.GetSimulatedStartUpPosition(0);
				N := N -1;
			END_FOR
			nCase := 120;
		
		120:	
			nActStopPos := UDINT_TO_UINT(nMoverCount-nNumMovers+1);
			FOR nForCounter:=1 TO nNumMovers DO
				fbMover[nForCounter].P_Dynamics.SetValuesVADJ(stMoverConfigNormal.velo,stMoverConfigNormal.Accel,stMoverConfigNormal.Decel,stMoverConfigNormal.Jerk);
				nMoveState[nForCounter] := 0;
				fbMover[nForCounter].MoveOnTrack(track:= GVL_Mc.MC_Tracks[E_TrackNum.Main], targetPos:= 300, gap:= stMoverConfigNormal.MoverGap);
			END_FOR

			nCase:= 130; 
		130:
			FOR nForCounter:=1 TO nMoverCount - (nMoverCount -nNumMovers)  DO
				CASE nMoveState[nForCounter] OF
					0:								
						IF Mover[nForCounter].MoverPos < 300 AND  Mover[nForCounter].TrackID = GVL_Mc.MC_Tracks[E_TrackNum.main].MCTOPLC_STD.TrackOID THEN
							fbMover[nForCounter].MoveOnTrack(track:= GVL_Mc.MC_Tracks[E_TrackNum.Main], targetPos:= aStopPositions[nActStopPos], gap:= stMoverConfigNormal.MoverGap);

							nActStopPos := nActStopPos + 1;
							nMoveState[nForCounter] := 10;
						END_IF
				END_CASE
			END_FOR
		
			bAllDone := TRUE;
			FOR nForCounter:=1 TO nNumMovers DO
				IF NOT(MoverFeedback[nForCounter].Done OR MoverFeedback[nForCounter].Error) THEN
					bAllDone := FALSE;
					EXIT;
				END_IF
			END_FOR
			
			IF bAllDone THEN
				nCase := 150;
			END_IF
		
		140:
			FOR nForCounter:=1 TO nNumMovers DO
				fbMover[nForCounter].P_PlanarMover.Halt(MoverFeedback[nForCounter], haltDynamics);
			END_FOR	
			
		nCase := 145;
			
		145:
			bAllDone := TRUE;
			FOR nForCounter:=1 TO nNumMovers DO
				IF NOT(MoverFeedback[nForCounter].Done OR MoverFeedback[nForCounter].Error) THEN
					bAllDone := FALSE;
					EXIT;
				END_IF
			END_FOR
			
			IF bAllDone THEN
				nCase := 150;
			END_IF
		
		//Disable
		150:

			FOR nForCounter:=1 TO nNumMovers DO
				fbMover[nForCounter].P_PlanarMover.Disable(MoverFeedback[nForCounter]);
			END_FOR
				
			nCase := 155;
		155:
			bAllDone := TRUE;
			FOR nForCounter:=1 TO nNumMovers DO
				IF NOT(MoverFeedback[nForCounter].Done OR MoverFeedback[nForCounter].Error) THEN
					bAllDone := FALSE;
					EXIT;
				END_IF
			END_FOR
			
			IF bAllDone THEN
				//MoverStopDone := TRUE;
				nCase := 0;
			END_IF	
END_CASE

bMagnetOn := FALSE;
FOR nForCounter:=1 TO nNumMovers DO
	IF  fbMover[nForCounter].XtsXlMover.GetPositionInfo_trackObjectId(0) = XtsShortcutOid THEN // this mover wll go through the switch start tracking his positon 
		switchingMoverPosition := fbMover[nForCounter].XtsXlMover.GetPositionInfo_trackPosition(0);  
	END_IF
	// check if the mover is in range of the switch position and on the switch track, if so turn on the magnet 
	IF fbMover[nForCounter].XtsXlMover.GetPositionInfo_trackObjectId(0) = XtsShortcutOid AND (IsBetween(fbMover[nForCounter].XtsXlMover.GetPositionInfo_trackPosition(0), SwitchConfig.MagnetStartPosition - (stMoverConfigNormal.Velo*0.045), SwitchConfig.MagnetEndPosition)) THEN
		bMagnetOn := TRUE; 
	END_IF
	moverInSwitch := nForCounter; 
END_FOR


IF SwitchConfig.UseNominalCurrentVeloSetpoints THEN
	SwitchStatus.CurrentTheorOutputMax := SwitchConfig.SwitchCurrentNominal;	
ELSE
	SwitchStatus.CurrentTheorOutputMax := ((SwitchConfig.DivertConfig.CurrentFunctionCoeffA*(((stMoverConfigNormal.Velo/1000)*(stMoverConfigNormal.Velo/1000))))+(SwitchConfig.DivertConfig.CurrentFunctionCoeffB*(stMoverConfigNormal.Velo/1000))+SwitchConfig.DivertConfig.CurrentFunctionCoeffC);	
END_IF

SwitchStatus.CurrentActualOutput := F_MapLReal(
	x:= MagnetFdbkValue, 
	in_min:= 0, 
	in_max:= 32767, 
	out_min:= 0, 
	out_max:= 54);

IF (nCase = 100) THEN
	IF bMagnetOn AND NOT Fault THEN
		MagnetValue := TO_INT(SwitchStatus.CurrentTheorOutputMax*1310);
	ELSE
		MagnetValue := 0;
	END_IF
ELSE // Manual Control of the Magnet Coil
	IF MagnetOnManHMICmd THEN
		MagnetValue := TO_INT(SwitchStatus.CurrentTheorOutputMax*1310);
	ELSE
		MagnetValue := 0;
		MagnetOnManHMICmd	:= FALSE;
	END_IF
END_IF


trapWhenMagnetturnedOn(CLK:= bMagnetOn); 
IF moverInSwitch <> 0 AND trapWhenMagnetTurnedOn.Q THEN 
	moverPositionWhenMagnetTurnedOn:=fbMover[moverInSwitch].XtsXlMover.GetPositionInfo_trackPosition(0);
END_IF


FP_Counter(clk:=bMagnetOn);

IF FP_Counter.Q THEN
	Switchcounter := Switchcounter+1;

END_IF



//distanceMonitoring of Mover 1 when on the big track 
IF Mover[1].TrackID = GVL_Mc.MC_Tracks[E_TrackNum.Main].MCTOPLC_STD.TrackOID THEN //calculate out how far it is to the mover in front 
	IF MOver[stMergeConfig.moverInFront].MoverPos -  Mover[1].MoverPos > 10 THEN 
		stMergeConfig.mover1FollowDist := MOver[stMergeConfig.moverInFront].MoverPos -  Mover[1].MoverPos;
	END_IF   
END_IF

END_PROGRAM

// ---- XlMover/POUs/FB_Mover.TcPOU
{attribute 'no_assign'}
FUNCTION_BLOCK FB_Mover IMPLEMENTS I_Mover
VAR_INPUT
END_VAR
VAR_OUTPUT
END_VAR
VAR
	_bIsInitialized: BOOL;	

	fbPlanarMover : MC_PlanarMover;
	fbPlanarFeedback: MC_PlanarFeedback;
	trackTrail: MC_PlanarTrackTrail;
	SyncMoverFeedback: Tc3_Mc3PlanarMotion.MC_PlanarFeedbackGearInPosOnTrackWithMasterMover;
	
	_GearInOptions: Tc3_Mc3PlanarMotion.ST_GearInPosOnTrackWithMasterMoverOptions;
	_stMoveOnTrackOptions: ST_MoveOnTrackOptions;
	_syncTrail : MC_PlanarTrackTrail;
	
	CmdFeedback :  XtsCommandFeedback;
	ipXtsMover:   I_XtsXlMover1;
	ipXtsProcessingUnit:  I_XtsProcessingUnit1;

	_stMoverInfos : ST_MoverInfo;	
	_stMoverOnTrackInfos : ST_MoverOnTrackInfo;

	_nextMcTrackOid: OTCID;
	_stDynamics: DynamicConstraint_PathXY;
	_TargetTrack : UDINT;
	_ReWork : BOOL;
	_partConfig: UINT;
	_InSync :BOOL; 
	_PositionOnTrack : LREAL;
	_Track : OTCID; 
	_distToEndOfTrack : LREAL;

	fbResult						: FB_TcMessage;
	_ipComObject					: ITComObject;
	PID_OnTrackInfos				: PTCID := 16#05030180;
	bInit 							: BOOL;
END_VAR

METHOD CycleUpdate : BOOL
VAR_INPUT
END_VAR
VAR 
	_trackEnum: e_TrackNum;
END_VAR
IF NOT _bIsInitialized THEN
	RETURN;
END_IF

fbPlanarMover.GetTrackTrailInformation(trackTrail);
_PositionOnTrack := fbPlanarMover.MCTOPLC.SETONTRACK.SetPos;
IF fbPlanarMover.MCTOPLC.SETONTRACK.TrackOID<>0 THEN 
	_Track := fbPlanarMover.MCTOPLC.SETONTRACK.TrackOID;
	_trackEnum := F_GetTrackEnum(fbPlanarMover.MCTOPLC.SETONTRACK.TrackOID); 
	_distToEndOfTrack := GVL_Mc.MC_Tracks[_trackEnum].GetLength()-_PositionOnTrack;
END_IF

fbPlanarMover.Update();

_stMoverinfos.MoverOtcid := fbPlanarMover.MCTOPLC.STD.MoverOID ;
_stMoverinfos.Positition :=	fbPlanarMover.MCTOPLC.SETONTRACK.SetPos;
_stMoverinfos.Track := fbPlanarMover.MCTOPLC.SETONTRACK.TrackOID;
_stMoverinfos.Error := fbPlanarMover.Error;
_stMoverinfos.ErrorID := fbPlanarMover.ErrorId;
_stMoverinfos.PlanarMoverCommandMode := fbPlanarMover.MCTOPLC.STD.CommandMode;
_stMoverinfos.State :=  fbPlanarMover.MCTOPLC.STD.State;
_stMoverinfos.Gap := _stMoverOnTrackInfos.Gap;
_stMoverinfos.LimitAcc := _stMoverOnTrackInfos.LimitA;
_stMoverinfos.LimitDec := _stMoverOnTrackInfos.LimitD;
_stMoverinfos.LimitJerk := _stMoverOnTrackInfos.LimitJ;
_stMoverinfos.LimitVelo := _stMoverOnTrackInfos.LimitV;
_stMoverinfos.TargetTrackPosition := _stMoverOnTrackInfos.TargetPosition;
_stMoverinfos.TargetTrack := _stMoverOnTrackInfos.TargetTrack;
_stMoverinfos.RemainingDistance := _stMoverOnTrackInfos.Remainingdistance;

fbPlanarFeedback.Update();
SyncMoverFeedback.Update(); 


UpdateXtsTrack();

GetOnTrackInfos();
END_METHOD

PROPERTY distToEndOfTrack : Lreal
GET
distToEndOfTrack := _distToEndOfTrack;
END_GET
END_PROPERTY

METHOD GetComObject : BOOL
VAR_INPUT
	nObjectId: OTCID;
END_VAR
IF FW_ObjMgr_GetObjectInstance(	oid		:= nObjectId, 
								iid		:= TC_GLOBAL_IID_LIST.IID_ITComObject, 
								pipUnk	:= ADR(_ipComObject)) = 0
THEN
	GetComObject := TRUE;
END_IF
END_METHOD

METHOD GetOnTrackInfos : BOOL
VAR
	nData 			: UDINT := SIZEOF(_stMoverOnTrackInfos);
	pData 			: PVOID := ADR(_stMoverOnTrackInfos);
	stEventEntry	: TcEventEntry;
	pstEventEntry	: REFERENCE TO TcEventEntry REF= stEventEntry;
END_VAR
VAR_INST
	hResult : HRESULT;
	bError : BOOL;
END_VAR
bError := FALSE;

IF _ipComObject <> 0 THEN 
	 hResult := 	_ipComObject.TcgetObjPara(		pid := PID_OnTrackInfos,
													nData := nData,
													pData := pData,
													pgp := 0); 	
	IF hResult = 0 THEN
		GetOnTrackInfos := TRUE;
	ELSE
		HRESULTAdsErr_TO_TcEventEntry(hResult,stEventEntry);
		IF NOT fbResult.EqualsToEventEntryEx( stOther := stEventEntry) THEN
			fbResult.CreateEx(stEventEntry, 0);
			fbResult.Send(0);
			fbResult.Release();
		END_IF
		bError := TRUE;
	END_IF							
END_IF
END_METHOD

METHOD Init : BOOL
VAR_INPUT

	XtsMover:   I_XtsXlMover1;
	XtsProcessingUnit :  I_XtsProcessingUnit1;
END_VAR



ipXtsMover:= XtsMover;
ipXtsProcessingUnit :=  XtsProcessingUnit;

_stMoveOnTrackOptions.direction := MC_Direction.mcDirectionPositive;
_stMoveOnTrackOptions.gapMode := MC_GAP_MODE_ON_TRACK.Fast1D;
_stMoveOnTrackOptions.gap:= 800;

_syncTrail.AddTrack(track:= GVL_Mc.MC_Tracks[E_TrackNum.Small]); 
_syncTrail.AddTrack(track:= GVL_Mc.MC_Tracks[E_TrackNum.Main]); 


//_stDynamics.SetValuesVADJ(500, 4000, 4000, 10000);

_bIsInitialized := TRUE;
Init := TRUE;


IF NOT bInit THEN
	IF GetComObject(nObjectId:=fbPlanarMover.MCTOPLC.STD.MoverOID) THEN
		bInit:=TRUE;
	END_IF
	RETURN;
END_IF
END_METHOD

METHOD JoinNearestTrack : BOOL


VAR_INST
	nForCounter: UINT;
	mcTrackOid: OTCID;
	partOid: OTCID;
	cmdFeedback					: 	XtsCommandFeedback;
	objectInfo: PlanarObjectInfo;
END_VAR
partOid := ipXtsMover.GetPositionInfo_partObjectId(cmdFeedback);

IF partOid = 0 THEN
	RETURN;
END_IF

IF cmdFeedback.IsDone THEN
	mcTrackOid := ipXtsProcessingUnit.XlPartWithOid(partOid, cmdFeedback).GetMcTrackOid(cmdFeedback);
	
	FOR nForCounter := 1 TO GVL_MC.nTrackCount DO
		objectInfo := GVL_MC.Mc_Tracks[nForCounter].GetPlanarObjectInfo();
		IF objectInfo.Id = mcTrackOid THEN
			fbPlanarMover.JoinTrack(fbPlanarFeedback, GVL_MC.Mc_Tracks[nForCounter], _stDynamics, 0); 
			RETURN;
		END_IF
	END_FOR
END_IF
END_METHOD

METHOD LeaveSystemAt : BOOL
VAR_INPUT
	ConnectionOut: REFERENCE TO MC_PlanarTrackConnectionOut;
END_VAR
fbPlanarMover.LeaveSystemAt(fbPlanarFeedback, ConnectionOut,  _stDynamics,0);
END_METHOD

METHOD MoveOnTrack : BOOL
VAR_INPUT
	track: REFERENCE TO MC_PlanarTrack;	
	targetPos: LREAL;
	gap : LREAL; 
END_VAR
_stMoveonTrackOptions.gap := gap; 

fbPlanarMover.MoveOnTrack(
	commandFeedback:= fbPlanarFeedback, 
	targetTrack:= track, 
	targetPositionOnTrack:= targetPos, 
	constraint:= _stDynamics, 
	options:= _stMoveOnTrackOptions);
END_METHOD

PROPERTY MoverOTCID : OTCID
GET
MoverOTCID := fbPlanarMover.MCTOPLC.STD.MoverOID;
END_GET
SET
END_SET
END_PROPERTY

PROPERTY MoverStopped : BOOL
GET
MoverStopped := (fbPlanarMover.MCTOPLC.SETONTRACK.SetVelo < 20);
END_GET
SET
END_SET
END_PROPERTY

PROPERTY P_Dynamics : REFERENCE TO DynamicConstraint_PathXY;
GET

P_Dynamics REF= _stDynamics;
END_GET
SET // PUBLIC
_stDynamics := P_Dynamics;
END_SET
END_PROPERTY

PROPERTY P_IsInitialized : bool
GET
P_IsInitialized := _bIsInitialized;
END_GET
END_PROPERTY

PROPERTY P_PlanarFeedback : REFERENCE TO MC_PlanarFeedback
GET
P_PlanarFeedback REF= fbPlanarFeedback;
END_GET
END_PROPERTY

PROPERTY P_PlanarMover :   REFERENCE TO  MC_PlanarMover
GET
P_PlanarMover REF= fbPlanarMover;
END_GET
END_PROPERTY

PROPERTY P_SyncFeedback :  REFERENCE TO MC_PlanarFeedbackGearInPosOnTrackWithMasterMover
GET
P_SyncFeedback REF= SyncMoverFeedback;
END_GET
END_PROPERTY

PROPERTY P_TargetTrack : UDINT
GET
P_TargetTrack := _TargetTrack ;
END_GET
SET
_TargetTrack := P_TargetTrack;
END_SET
END_PROPERTY

PROPERTY Rework : BOOL
GET
Rework := _Rework;
END_GET
SET
_Rework := Rework;
END_SET
END_PROPERTY

METHOD SyncToOtherMover : BOOL
VAR_INPUT
	masterSyncPos : LREAL; // Position on the master track
	followerSyncPos : LREAL; // position on the follower track
	PlanarMoverToFollow: REFERENCE TO Tc3_Mc3PlanarMotion.MC_PlanarMover;
	masterTrack : REFERENCE TO Tc3_Mc3PlanarMotion.MC_PlanarTrack; 
	followerTrack : REFERENCE TO Tc3_Mc3PlanarMotion.MC_PlanarTrack; 
	velo : REFERENCE TO LREAL; 
END_VAR

VAR
	trail: Tc3_Mc3PlanarMotion.MC_PlanarTrackTrail;

END_VAR
_GearInOptions.allowedSlaveSyncDirections := MC_SYNC_DIRECTIONS.Positive; 
_GearInOptions.directionMasterSyncPosition := MC_DIRECTION.mcDirectionNonModulo; 
_GearInOptions.directionSlaveSyncPosition := MC_DIRECTION.mcDirectionNonModulo;  
_GearInOptions.followMover := FALSE; 
_GearInOptions.gap := 0; // elimnate gap funciton 
_GearInOptions.inSyncToleranceDistance :=0; 
_GearInOptions.moduloToleranceMasterSyncPosition := 0; 
_GearInOptions.moduloToleranceSlaveSyncPosition := 0;  
_stDynamics.V := velo; 

fbPlanarMover.GearInPosOnTrackWithMasterMover(
	commandFeedback:=  SyncMoverFeedback , 
	masterMover:= PlanarMoverToFollow , 
	trackTrail:= _syncTrail, // may need to give a trail maybe not
	masterSyncPosition:= masterSyncPos, 
	masterSyncPositionTrack:= MasterTrack , 
	slaveSyncPosition:= followerSyncPos, 
	slaveSyncPositionTrack:= followerTrack, 
	constraint:=_stDynamics , 
	options:=_GearInOptions );
END_METHOD

METHOD PUBLIC UpdateXtsTrack
VAR_INPUT
END_VAR
VAR_STAT
	nTrackCount: UINT;
	oid1: OTCID;
	oid2: OTCID;
	
	nForCounter: UINT;
	nPartConfigCount: UINT;
	
	partConfig1: OTCID;
	partConfig2: OTCID;
	
	mcTrackOid1: OTCID;
	mcTrackOid2: OTCID;
	trackOid: OTCID;
	
	nTrackTrailCount: UDINT;
	actTrackOid: OTCID;
	nIndexInTrail: UDINT;
END_VAR
nTrackTrailCount := trackTrail.TrackCount;
actTrackOid := fbPlanarMover.MCTOPLC.SETONTRACK.TrackOID;

IF nTrackTrailCount <= 1 THEN
	RETURN;
END_IF

FOR nForCounter := 1 TO UDINT_TO_UINT(nTrackTrailCount) DO
	oid1 := trackTrail.GetTrackOidAt(nForCounter);
	IF oid1 = actTrackOid THEN
		IF nForCounter < nTrackTrailCount THEN
			oid2 := trackTrail.GetTrackOidAt(nForCounter + 1);
			EXIT;
		ELSE
			RETURN; //last one ine track trail
		END_IF
	END_IF
END_FOR

IF oid2 = _nextMcTrackOid AND   ipXtsMover.GetPositionInfo_partPosition(CmdFeedback) < 600THEN //no change
	RETURN;
END_IF

nTrackCount := ipXtsProcessingUnit.TrackCount();

FOR nForCounter := 1 TO nTrackCount DO
	nPartConfigCount := ipXtsProcessingUnit.Track(nForCounter, CmdFeedback).PartConfigCount(); 
	
	IF nPartConfigCount >= 2  THEN
		partConfig1 := ipXtsProcessingUnit.Track(nForCounter, CmdFeedback).GetPartConfigOidAt(1, 0);
		partConfig2 := ipXtsProcessingUnit.Track(nForCounter, CmdFeedback).GetPartConfigOidAt(2, 0);
//
		
		IF partConfig1 = 0 OR partConfig2 = 0 THEN
			CONTINUE;
		END_IF
		
		mcTrackOid1 := ipXtsProcessingUnit.XlPartWithOid(partConfig1, CmdFeedback).GetMcTrackOid(0);
		mcTrackOid2 := ipXtsProcessingUnit.XlPartWithOid(partConfig2, CmdFeedback).GetMcTrackOid(0);
		IF mcTrackOid1 = oid1 AND mcTrackOid2 = oid2   THEN
			trackOid := ipXtsProcessingUnit.Track(nForCounter, CmdFeedback).GetObjectId();
			ipXtsMover.SetActiveTrackObjectId(trackOid, CmdFeedback);
			
			IF CmdFeedback.IsDone THEN
				_nextMcTrackOid := oid2;
			END_IF
			
			RETURN;
		END_IF
	END_IF
END_FOR
END_METHOD

PROPERTY XlProcessingUnit : I_XtsProcessingUnit1
GET
XlProcessingUnit := ipXtsProcessingUnit;
END_GET
END_PROPERTY

PROPERTY XtsComFeed : REFERENCE TO  XtsCommandFeedback
GET
XtsComFeed REF= CmdFeedback;
END_GET
END_PROPERTY

PROPERTY XtsXlMover : I_XtsXlMover1
GET
XtsXlMover := ipXtsMover;
END_GET
END_PROPERTY

END_FUNCTION_BLOCK
